// TIA Portal V16 export
// export: Created 2026-06-18T08:15:20.5409663Z, ExportSetting WithDefaults, DisplayName Totally Integrated Automation Portal, DisplayVersion V16 Update 8, DisplayName TIA Portal Version Control Interface, DisplayVersion V16 Update 8, DisplayName TIA Portal Openness, DisplayVersion V16 Update 8, DisplayName SINAMICS Startdrive Advanced, DisplayVersion V16, DisplayName SINAMICS Startdrive G130, G150, S120, S150, SINAMICS MV, S210, DisplayVersion V16, DisplayName SINAMICS Startdrive G110M, G120, G120C, G120D, G120P, DisplayVersion V16, DisplayName STEP 7 Professional, DisplayVersion V16 Update 8, DisplayName STEP 7 Safety, DisplayVersion V16 Update 7, DisplayName WinCC Advanced, DisplayVersion V16 Update 8
Screen "Temp_Monitor"  800x480, Number=1
  ScreenLayer 
    IOField "IO_Temp1" at 180,85 size 100x40  DataFormat=Decimal, FormatPattern=9999999, Mode=InOutput
    IOField "IO_Temp3" at 180,225 size 100x40  DataFormat=Decimal, FormatPattern=9999999, Mode=InOutput
    IOField "IO_Temp2" at 180,155 size 100x40  DataFormat=Decimal, FormatPattern=9999999, Mode=InOutput
    SymbolicIOField "SIO_Status" at 120,340 size 120x40  CountVisibleItems=3, Mode=InOutput, OnValue=1, TextOff="0", TextOn="1"
    TextField "TXT_Title" at 260,20 size 280x40  Text="温度监控画面"
    TextField "TXT_StatusLabel" at 30,340 size 80x40  Text="系统状态"
    Button "BTN_ResetAlarm" at 400,340 size 120x50  Mode=Text, TextOff="复位报警", TextOn="复位报警"
    Circle "LMP_Alarm1" at 340,85 size 48x48
    Circle "LMP_Alarm3" at 340,225 size 48x48
    Circle "LMP_Alarm2" at 340,155 size 48x48
